PROGRAM OP20_ERROR
VAR
	OP20_StErr_1: TON;
	OP20_Step_Err_2: TON;
	OP20_StepErr_3: TON;
	OP20_StErr_4: TON;
	OP20_Step_Err_5: TON;
	OP20_StepErr_6: TON;
//	end: INT;
END_VAR


//Reset ErrorActive
IF (OP20_HMI_Reset OR Servo_Reset) THEN 
	OP20_GVL.OP20_ErrorActive:= FALSE;
	OP20_GVL.OP20_ErrorWord_0:= 0;
	OP20_GVL.OP20_ErrorWord_1:= 0;
	OP20_GVL.OP20_ErrorWord_2:= 0;	
END_IF

//(OP20_GVL.OP20_ErrorWord_0<>0) OR
// Set ERROR ACTIVE
IF ( (OP20_GVL.OP20_ErrorWord_1<>0) OR (OP20_GVL.OP20_ErrorWord_2<>0)) THEN
	OP20_GVL.OP20_ErrorActive:= TRUE;
END_IF


OP20_ErrorWord_0.0:= SR20_Vert_servo_ctrl.Axis_Error;
OP20_ErrorWord_0.1:= NOT OperationEnable;
// Auto Seq Step Error
//Servo not reaching work position
OP20_StErr_1(IN:=(OP20_GVL.OP20_AUTO_STP_NO=80) , PT:=T#5S , Q=> , ET=> );
IF (OP20_GVL.OP20_AUTO_STP_NO=80 AND NOT OP20_GVL.OP20_SERVO_ON_WRK AND OP20_StErr_1.Q) THEN
	OP20_GVL.OP20_ErrorWord_0.2:=TRUE;
END_IF

// Servo Not Reached home position or safe-work position
OP20_Step_Err_2(IN:=OP20_GVL.OP20_AUTO_STP_NO=160, PT:=T#5S , Q=> , ET=> );
IF (OP20_GVL.OP20_AUTO_STP_NO=160 AND NOT OP20_SERVO_ON_SFE_WRK AND OP20_Step_Err_2.Q) THEN
	OP20_GVL.OP20_ErrorWord_0.3:=TRUE;
END_IF
OP20_GVL.OP20_ErrorWord_0.4:=0;
//OP20_StepErr_3(IN:=( OP20_HomeRunning AND (OP20_Homing_Seq=10) AND NOT SR20_Vert_servo_ctrl.Axis_In_Home), PT:=T#10S , Q=> , ET=> );
//IF OP20_StepErr_3.Q THEN
//	OP20_GVL.OP20_ErrorWord_0.4:=TRUE;
//END_IF

END_PROGRAM

(* stored: Version 1.1.0.1, ProductVersion 3.1.4024.11
   POU OP20_ERROR: Id {c2fb98fc-474d-4f41-b7d0-86b62e4f094a}, SpecialFunc None *)
